# EPICS substitutions: evrseqcalcApp/Db/evrseqcalc.substitutions
file evrcalcdelay.template
{
pattern {SYS, DEV, EVR}
	{$(SYS_EVRSEQ), $(DEV1), $(EVR_EVRSEQ)}
	{$(SYS_EVRSEQ), $(DEV2), $(EVR_EVRSEQ)}
	{$(SYS_EVRSEQ), $(DEV3), $(EVR_EVRSEQ)}
	{$(SYS_EVRSEQ), $(DEV4), $(EVR_EVRSEQ)}
}

file asubevrseq.template
{
pattern {SYS, EVR}
	{$(SYS_EVRSEQ), $(EVR_EVRSEQ)}
}
